// TwinCAT 3 PLC project Nepionic_Log_Syslog
// Title: Nepionic_Log_Syslog
// Company: Nepionic
// Author: Nepionic
// ProjectVersion: 0.1.0
// ProgramVersion: 3.1.4026.21
// libraries:
//   [Nepionic_Log], * (Nepionic)
//   Tc2_Standard, * (Beckhoff Automation GmbH)
//   Tc2_System, * (Beckhoff Automation GmbH)
//   Tc2_TcpIp, * (Beckhoff Automation GmbH)
//   Tc2_Utilities, * (Beckhoff Automation GmbH)
// project tree:
//   Lib/ SyslogAppender.TcPOU, SyslogClient.TcPOU

// ---- Lib/SyslogAppender.TcPOU
{attribute 'linkalways'}
{attribute 'no_explicit_call' := 'This FB is a CLASS and must be accessed using methods or properties'}
{attribute 'enable_dynamic_creation'}
/// Syslog (RFC 5424, UDP) log appender for Nepionic_Log.
/// Implements `LogAppender` by forwarding records to a `SyslogClient` that
/// transmits them over UDP.
///
/// **Important:** `Execute` must be called once each PLC cycle to drive the
/// underlying UDP state machine:
/// ```st
/// // In your cyclic PROGRAM:
/// syslog_appender.Execute();
/// ```
///
/// Usage (startup):
/// ```st
/// GetLogManager().Register(syslog_appender);
/// ```
///
/// Structured attributes are appended to the syslog message body as
/// `key=value` pairs separated by spaces. They are not encoded as RFC 5424
/// structured data.
FUNCTION_BLOCK PUBLIC SyslogAppender IMPLEMENTS Nepionic_Log.LogAppender
VAR
	client : SyslogClient(hostname := '127.0.0.1', port := 514);
	_level : Nepionic_Log.LogLevel := Nepionic_Log.LogLevel.Debug;
END_VAR

METHOD PUBLIC Append : BOOL
VAR_INPUT
	level : Nepionic_Log.LogLevel;
	message : Tc2_System.T_MaxString;
	source : Tc2_System.T_MaxString;
	attributes : ARRAY[0..9] OF Nepionic_Log.LogAttribute;
	attribute_count : USINT;
END_VAR
VAR
	syslog_severity : INT;
	text : STRING(255);
	i : USINT;
END_VAR
CASE level OF
	Nepionic_Log.LogLevel.Debug:       syslog_severity := 7;
	Nepionic_Log.LogLevel.Information: syslog_severity := 6;
	Nepionic_Log.LogLevel.Warning:     syslog_severity := 4;
	Nepionic_Log.LogLevel.Error:       syslog_severity := 3;
	Nepionic_Log.LogLevel.Fatal:       syslog_severity := 2;
ELSE
	syslog_severity := 6;
END_CASE

// Build message: "[source] message  key=value key=value"
IF Tc2_Standard.Len(source) > 0 THEN
	text := Tc2_Standard.Concat('[', Tc2_Standard.Concat(source, '] '));
END_IF
text := Tc2_Standard.Concat(text, message);

IF attribute_count > 0 THEN
	FOR i := 0 TO attribute_count - 1 DO
		text := Tc2_Standard.Concat(text, ' ');
		text := Tc2_Standard.Concat(text, Tc2_Standard.Concat(attributes[i].key, Tc2_Standard.Concat('=', Nepionic_Log.LogAttributeValueToString(attributes[i]))));
	END_FOR
END_IF
client.SendLog(syslog_severity, text);
Append := TRUE;
END_METHOD

/// Application name embedded in the syslog header (default `TwinCAT_PLC`).
{attribute 'monitoring' := 'call'}
PROPERTY PUBLIC AppName : STRING(32)
GET // PUBLIC
AppName := client.AppName;
END_GET
SET // PUBLIC
client.AppName := AppName;
END_SET
END_PROPERTY

/// Drive the underlying UDP state machine.
/// Must be called once each PLC cycle.
METHOD PUBLIC Execute
client.Execute();
END_METHOD

METHOD FB_Init : BOOL
VAR_INPUT
	bInitRetains : BOOL;
	bInCopyCode : BOOL;
	/// IP address or hostname of the syslog server.
	hostname : STRING(15) := '127.0.0.1';
	/// UDP port of the syslog server (default 514).
	port : UINT := 514;
END_VAR
client.Hostname := hostname;
client.Port := port;
END_METHOD

{attribute 'monitoring' := 'call'}
PROPERTY PUBLIC Level : Nepionic_Log.LogLevel
GET // PUBLIC
Level := _level;
END_GET
SET // PUBLIC
_level := Level;
END_SET
END_PROPERTY

END_FUNCTION_BLOCK

// ---- Lib/SyslogClient.TcPOU
{attribute 'linkalways'} 
{attribute 'no_explicit_call' := 'This FB is a CLASS and must be accessed using methods or properties'}
{attribute 'enable_dynamic_creation'}
FUNCTION_BLOCK PUBLIC SyslogClient
VAR
	// Properties
	_hostname : STRING := '127.0.0.1';
	_port : UINT := 514;
	app_name : STRING(32) := 'TwinCAT_PLC';
    
	// Internal Logic
	socket_handle : Tc2_TcpIp.T_HSocket;
	socket_create : Tc2_TcpIp.Fb_SocketUdpCreate;
	udp_send : Tc2_TcpIp.Fb_SocketUdpSendTo;
    
	log_payload : STRING(512);
	timestamp : STRING(32);
	get_time : Tc2_Utilities.NT_GetTime;
    
	state : INT := 0;
END_VAR

PROPERTY PUBLIC AppName : STRING(255)
GET // PUBLIC
AppName := app_name;
END_GET
SET // PUBLIC
app_name := AppName;
END_SET
END_PROPERTY

METHOD PUBLIC Execute
CASE state OF
    0: // Idle
        
    10: // Fetch Timestamp
        get_time(START := TRUE);
        IF NOT get_time.BUSY AND NOT get_time.ERR THEN
            UpdateTimestamp();
            get_time(START := FALSE);
            state := 20;
        ELSIF get_time.ERR THEN
            get_time(START := FALSE);
            state := 0;
        END_IF

    20: // Maintain Socket
        IF socket_handle.handle = 0 THEN
			socket_create(
				bExecute := TRUE,
				sLocalHost := _hostname,
				nLocalPort := 4444
			);
			IF NOT socket_create.bBusy AND NOT socket_create.bError THEN
				socket_handle := socket_create.hSocket;
				socket_create(bExecute := FALSE);
			END_IF
		ELSE
			state := 30;
		END_IF

    30: // Dispatch UDP
        udp_send(
            hSocket := socket_handle, 
            sRemoteHost := _hostname, 
            nRemotePort := _port,
            pSrc := ADR(log_payload), 
            cbLen := INT_TO_UDINT(Tc2_Standard.Len(log_payload)), 
            bExecute := TRUE
		);
            
        IF NOT udp_send.bBusy AND NOT udp_send.bError THEN
            udp_send(bExecute := FALSE);
            state := 0; 
        END_IF
END_CASE
END_METHOD

//FB_Init is always available implicitly and it is used primarily for initialization.
//The return value is not evaluated. For a specific influence, you can also declare the
//methods explicitly and provide additional code there with the standard initialization
//code. You can evaluate the return value.
METHOD FB_Init: BOOL
VAR_INPUT
	bInitRetains: BOOL; // TRUE: the retain variables are initialized (reset warm / reset cold)
	bInCopyCode: BOOL;  // TRUE: the instance will be copied to the copy code afterward (online change)
	hostname : STRING(15) := '127.0.0.1';
	port : UINT := 514;
END_VAR
THIS^._hostname := hostname;
THIS^._port := port;
END_METHOD

PROPERTY PUBLIC Hostname : STRING(15)
GET // PUBLIC
Hostname := _hostname;
END_GET
SET // PUBLIC
_hostname := Hostname;
ResetConnection();
END_SET
END_PROPERTY

PROPERTY PUBLIC Port : UINT
GET // PUBLIC
Port := _port;
END_GET
SET // PUBLIC
_port := Port;
ResetConnection();
END_SET
END_PROPERTY

METHOD PRIVATE ResetConnection
END_METHOD

METHOD PUBLIC SendLog
VAR_INPUT
	severity : INT; // 0: Emerg ... 7: Debug
	message  : STRING(255);
END_VAR
VAR_INST
	priority : INT;
END_VAR
// Facility 1 (User) * 8 + severity
priority := 8 + severity;

// Build RFC 5424 String: <PRI>1 TIMESTAMP HOSTNAME APPNAME - - - MESSAGE
log_payload := Tc2_System.Concat('<', INT_TO_STRING(priority));
log_payload := Tc2_System.Concat(log_payload, '>1 ');
log_payload := Tc2_System.Concat(log_payload, timestamp);
log_payload := Tc2_System.Concat(log_payload, ' ');
log_payload := Tc2_System.Concat(log_payload, hostname);
log_payload := Tc2_System.Concat(log_payload, ' ');
log_payload := Tc2_System.Concat(log_payload, app_name);
log_payload := Tc2_System.Concat(log_payload, ' - - - ');
log_payload := Tc2_System.Concat(log_payload, message);

state := 10;
END_METHOD

METHOD PRIVATE UpdateTimestamp
timestamp := WORD_TO_STRING(get_time.TimeStr.wYear);
timestamp := Tc2_System.Concat(timestamp, '-');
timestamp := Tc2_System.Concat(timestamp, Tc2_System.Right(Tc2_System.Concat('0', WORD_TO_STRING(get_time.TimeStr.wMonth)), 2));
timestamp := Tc2_System.Concat(timestamp, '-');
timestamp := Tc2_System.Concat(timestamp, Tc2_System.Right(Tc2_System.Concat('0', WORD_TO_STRING(get_time.TimeStr.wDay)), 2));
timestamp := Tc2_System.Concat(timestamp, 'T');
timestamp := Tc2_System.Concat(timestamp, Tc2_System.Right(Tc2_System.Concat('0', WORD_TO_STRING(get_time.TimeStr.wHour)), 2));
timestamp := Tc2_System.Concat(timestamp, ':');
timestamp := Tc2_System.Concat(timestamp, Tc2_System.Right(Tc2_System.Concat('0', WORD_TO_STRING(get_time.TimeStr.wMinute)), 2));
timestamp := Tc2_System.Concat(timestamp, ':');
timestamp := Tc2_System.Concat(timestamp, Tc2_System.Right(Tc2_System.Concat('0', WORD_TO_STRING(get_time.TimeStr.wSecond)), 2));
timestamp := Tc2_System.Concat(timestamp, 'Z');
END_METHOD

END_FUNCTION_BLOCK
